(* CODESYS project simulacoes.project

Project tree, tasks and I/O mapping:
  Device : CODESYS Control Win V3, 3S - Smart Software Solutions GmbH, version 3.5.12.10
    application Application
      libraries: VisuDialogs, * (System); Util, * (System); Standard, * (System)
      task DefaultTask (cyclic, interval T#10ms, priority 16) calls PLC_PRG
      Data types/
      Global Variables/
        global variables ParafusosIOs
        global variables GVL
      POUs/
        program PLC_PRG [ST]
      Visualizations/
        visualisation tanque_DIG
        visualisation SILO
        visualisation semaforo
        visualisation garagem
        visualisation tanque_ANALOG
      trace Sampling_Trace (task ): 
      PROGRAMAS/
        garagem/
          program garagem_LD [LD]
          program garagem_ST [ST]
        tanqueD/
          program tanqueD_batelada [ST]
          program tanqueD_auto [ST]
          program tanqueD_main [ST]
          program tanqueD_manual [ST]
        silo/
          program silo_LD [LD]
          program silo_ST [ST]
        semaforo/
          program semaforo_LD [LD]
          program semaforo_ST [ST]
        tanqueA/
          program tanqueA_main [ST]
          function VOL_TO_LEVEL [ST]
          program tanqueA_process [ST]
          program tanqueA_manut [ST]
      SIMULADORES/
        program SIM_GARAGEM [LD]
        program SIM_SILO [LD]
        program SIMULADORES [ST]
        program SIM_TANQUE_DIG [LD]
        program SIM_TANQUE_ANALOG [LD]
      image pool ImagePool
      Symbols
  libraries: Standard, 3.5.12.0 (System); IecSfc, 3.4.2.0 (System); SysCallback23, 3.5.2.0 (System); VisuSymbols, 3.5.10.0 (System)
  GlobalImagePool
  text list GlobalTextList
  5ce3da45-db07-42e7-a21c-a00fff4ed8f6|semaforo\WALK2.bmp
*)

// Device/Application/Global Variables/ParafusosIOs
VAR_GLOBAL
// I/Os - SILO
	// Entradas digitais:
		xParBStartSilo	 :	BOOL;
		xParBStopSilo	 :	BOOL;
		xParChASilo		 :	BOOL;
		xParChBSilo		 :	BOOL;
		xParChCSilo		 :	BOOL;
		xParLevel				  :	BOOL;
		xParProx 				  :	BOOL;
	// Saídas digitais:
		xParRunSilo		 : BOOL;
		xParFillSilo	 : BOOL;
		xParFullSilo	 : BOOL;
		xParValve 		 : BOOL;
		xParMotor 		 : BOOL;

// I/Os - Semáforo
	// Entradas digitais:
		xParafBPedE 	 :	BOOL;
		xParafBPedD 	 :	BOOL;
	// Saídas digitais:
		xParafVermE 	 : BOOL;
		xParafVermD 	 : BOOL;
		xParafVerdE 	 : BOOL;
		xParafVerdD		 : BOOL;
		xParafAmarE 	 : BOOL;
		xParafAmarD 	 : BOOL;

// I/Os - Garagem
	// Entradas digitais:
		xParBOpen 		          :	BOOL;
		xParBClose 		 :	BOOL;
		xParBStopGar	 :	BOOL;
		xParLs1 		 		  :	BOOL;
		xParLs2 		  		  :	BOOL;
	// Saídas digitais:
		xParAjar		 : BOOL;
		xParOpen 		 : BOOL;
		xParShut 		 : BOOL;
		xParMotorUp 	 : BOOL;
		xParMotorDown	 : BOOL;

// I/Os - Tanque (Digital)
	// Entradas digitais:
		xParBStartTankD	 :	BOOL;
		xParBStopTankD	 :	BOOL;
		xParChATankD	 :	BOOL;
		xParChBTankD	 :	BOOL;
		xParChCTankD	 :	BOOL;
		xParFluxo1				  :	BOOL;
		xParFluxo2				  :	BOOL;
		xParFluxo3				  :	BOOL;
		xParTermostato			  :	BOOL;
		xParAltoD				  :	BOOL;
		xParBaixoD				  :	BOOL;
	// Saídas digitais:	
		xParBomba1D		 : BOOL;
		xParBomba2D		 : BOOL;
		xParBomba3D		 : BOOL;
		xParAquecD		 : BOOL;
		xParMistD		 : BOOL;
		xParRunTankD	 : BOOL;
		xParFullTankD	 : BOOL;
		xParIdleD		 : BOOL;

// I/Os - Tanque (Analógico)
	// Entradas digitais:
		xParBStartTankA	 :	BOOL;
		xParBStopTankA	 :	BOOL;
		xParChATankA	 :	BOOL;
		xParChBTankA	 :	BOOL;
		xParChCTankA	 :	BOOL;	
	// Entradas analógicas:
		iParSPB1				  :	INT;
		iParSPB2	 			  :	INT;
		iParSPTemp				  :	INT;
		iParUltras				  :	INT;
		iParTerm				  :	INT;
	// Saídas digitais:	
		xParBomba1A		 : BOOL;
		xParBomba2A		 : BOOL;
		xParBomba3A		 : BOOL;
		xParAquecA		 : BOOL;
		xParMistA		 : BOOL;
		xParRunTankA	 : BOOL;
		xParFullTankA	 : BOOL;
		xParIdleA		 : BOOL;
	// Saidas analógicas:	
		iParDisplayTemp    : INT;
		iParDisplayNivel   : INT;
END_VAR

// Device/Application/Global Variables/GVL
VAR_GLOBAL
	l1 : REAL := 2000.0;
	l2 : REAL := 5000.0;
	k : REAL := (10000.0/64.0); //Constante de conversão (litros/pulso)
	TankDMode : INT := 0;
	xEnableTankD : BOOL;
	LimTankD : REAL;
	xEnableTankA : BOOL;
	iTankAUnit : INT;
	TankAMode : INT := 0;
	rSupI1 : REAL;
	rSupI2 : REAL;
	rSupT : REAL;
	rTankALevel : REAL;
	rTankATemp : REAL;
	xTankARunning : BOOL;
	rTankASP1 : REAL;
	rTankASP2 : REAL;
	rTankASPTemp : REAL;
	allowStart : BOOL;
	LimTankA : REAL;
	blinkEnable : BOOL;
	blinkDuration : INT;
	tonoff : REAL;
	NULL : BOOL := FALSE;
	blinkTarget : POINTER TO BOOL := ADR(NULL);
	halfCicle : BOOL;
	heat : BOOL;
	LimTankAConv : REAL;
	capMax : REAL;
	defaultUnit : INT;
	rTankAVol : REAL;
	offset : REAL;
	batCont : INT := 0;
	prod : REAL := 0;
	processTarget : INT := 0;
	xEndLess : BOOL := TRUE;
	processID : INT;
	xstopAfterCurrent : BOOL;
	rTankDVol : REAL;
END_VAR

// Device/Application/POUs/PLC_PRG
PROGRAM PLC_PRG
VAR

END_VAR

SIMULADORES();
//garagem_LD();
garagem_ST();
//silo_LD();
silo_ST();
//semaforo_LD();
semaforo_ST();
tanqueD_main();
tanqueA_main();

END_PROGRAM

// Device/Application/SIMULADORES/SIMULADORES
PROGRAM SIMULADORES
VAR
END_VAR

SIM_GARAGEM();
SIM_SILO();
SIM_TANQUE_DIG();
SIM_TANQUE_ANALOG();

END_PROGRAM

// Device/Application/SIMULADORES/SIM_GARAGEM
PROGRAM SIM_GARAGEM
VAR
	portao		: 	RAMP_INT;
	porta		: 	INT;
	pin			: 	INT;
	T2g		: 	TON;
	T1g		: 	TON;
	fogo		: 	BOOL;
	fechado	: 	BOOL;
	aberto		: 	BOOL;
	Tfogo		: 	TON;
	fogosobe	: 	BOOL;
	fogodesce: 	BOOL;
	Pisca: BOOL;
	Pisca1: BLINK;
END_VAR
VAR // added by the converter: edge detectors and wires of the graphical bodies
    _w1 : USINT;
    _w2 : INT;
END_VAR

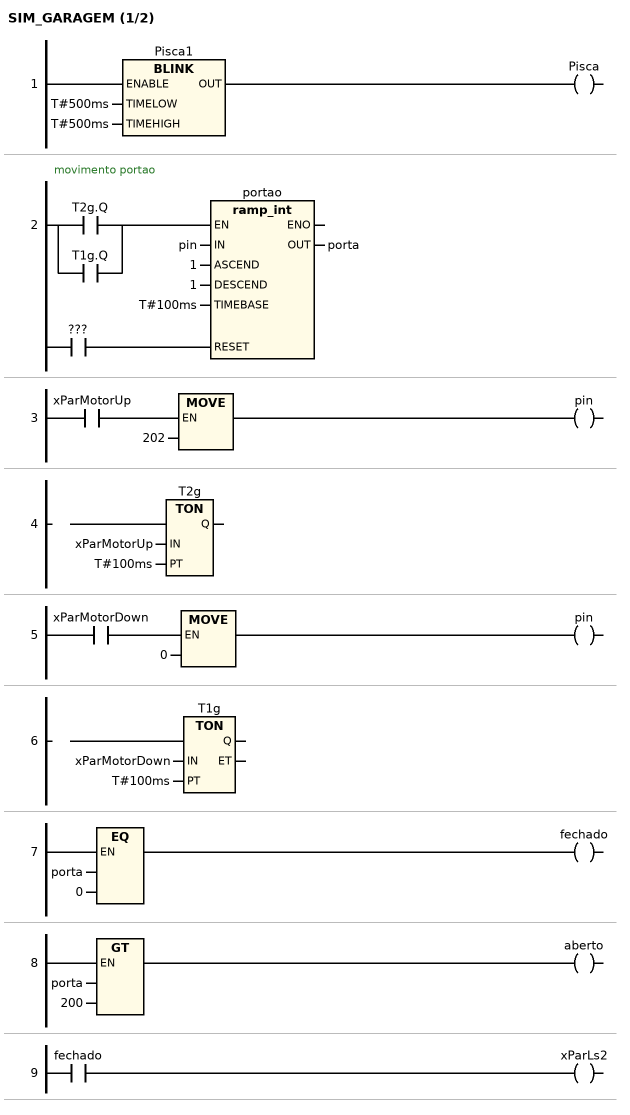
// NETWORK 1
Pisca1(ENABLE := TRUE, TIMELOW := T#500ms, TIMEHIGH := T#500ms); // BLINK
Pisca := Pisca1.OUT;

// NETWORK 2
// movimento portao
IF T2g.Q OR T1g.Q THEN
    portao(IN := pin, ASCEND := 1, DESCEND := 1, TIMEBASE := T#100ms, OUT => porta); // ramp_int
END_IF

// NETWORK 3
IF xParMotorUp THEN _w1 := 202; END_IF
pin := _w1;

// NETWORK 4
T2g(IN := xParMotorUp, PT := T#100ms); // TON

// NETWORK 5
IF xParMotorDown THEN _w2 := 0; END_IF
pin := _w2;

// NETWORK 6
T1g(IN := xParMotorDown, PT := T#100ms); // TON

// NETWORK 7
fechado := porta = 0;

// NETWORK 8
aberto := porta > 200;

// NETWORK 9
xParLs2 := fechado;

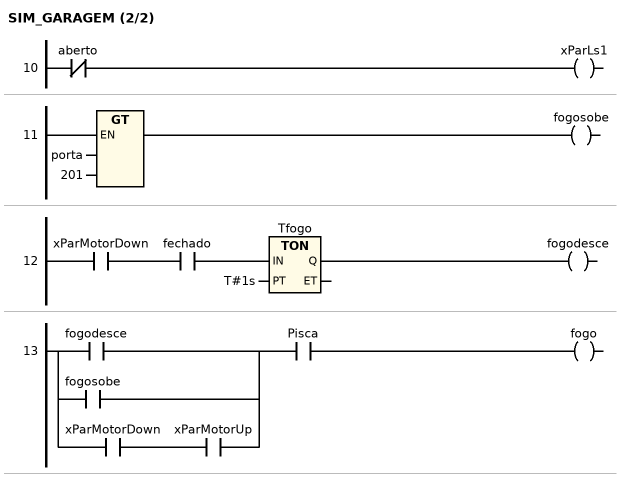
// NETWORK 10
xParLs1 := NOT aberto;

// NETWORK 11
fogosobe := porta > 201;

// NETWORK 12
Tfogo(IN := xParMotorDown AND fechado, PT := T#1s); // TON
fogodesce := Tfogo.Q;

// NETWORK 13
fogo := (fogodesce OR fogosobe OR xParMotorDown AND xParMotorUp) AND Pisca;

END_PROGRAM

// Device/Application/SIMULADORES/SIM_SILO
PROGRAM SIM_SILO
VAR
	aaux			: 	BOOL;
	Tcx				: 	TON;
	ccx				: 	CTU;
	resetesteira	: 	BOOL;
	caixa_mov1	: 	INT;
	caixa_mov		: 	INT;
	prox1			: 	BOOL;
	prox2			: 	BOOL;
	Tlevel			: 	TON;
	clevel			: 	CTU;
	level1			: 	INT;
	auxlevel		: 	BOOL;
	Talaga			: 	TON;
	calaga			: 	CTU;
	alaga			: 	INT;
	RESET		: 	BOOL;
	Pisca: BOOL;
	Pisca1: BLINK;
	CHEIA: BOOL;
END_VAR

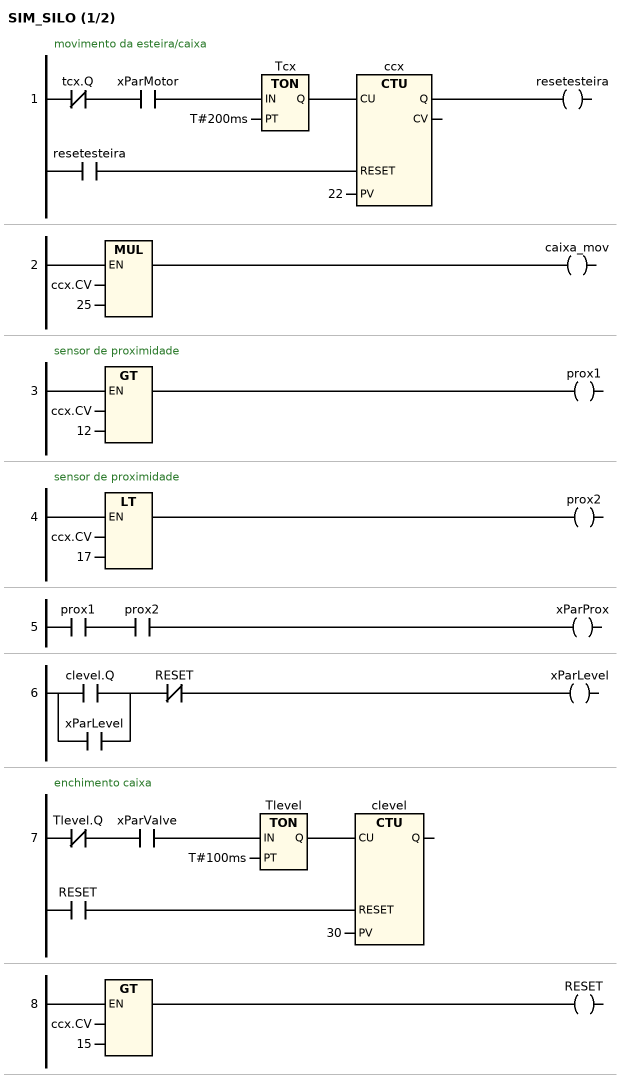
// NETWORK 1
// movimento da esteira/caixa
Tcx(IN := NOT tcx.Q AND xParMotor, PT := T#200ms); // TON
ccx(CU := Tcx.Q, RESET := resetesteira, PV := 22); // CTU
resetesteira := ccx.Q;

// NETWORK 2
caixa_mov := ccx.CV * 25;

// NETWORK 3
// sensor de proximidade
prox1 := ccx.CV > 12;

// NETWORK 4
// sensor de proximidade
prox2 := ccx.CV < 17;

// NETWORK 5
xParProx := prox1 AND prox2;

// NETWORK 6
xParLevel := (clevel.Q OR xParLevel) AND NOT RESET;

// NETWORK 7
// enchimento caixa
Tlevel(IN := NOT Tlevel.Q AND xParValve, PT := T#100ms); // TON
clevel(CU := Tlevel.Q, RESET := RESET, PV := 30); // CTU

// NETWORK 8
RESET := ccx.CV > 15;

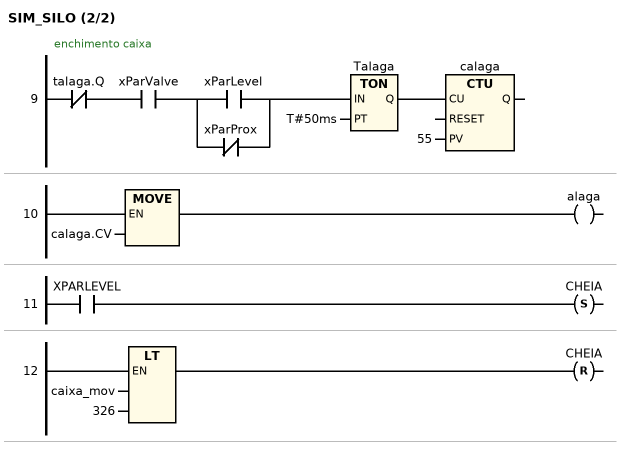
// NETWORK 9
// enchimento caixa
Talaga(IN := NOT talaga.Q AND xParValve AND (xParLevel OR NOT xParProx), PT := T#50ms); // TON
calaga(CU := Talaga.Q, PV := 55); // CTU

// NETWORK 10
alaga := calaga.CV;

// NETWORK 11
CHEIA S= XPARLEVEL;

// NETWORK 12
CHEIA R= caixa_mov < 326;

END_PROGRAM

// Device/Application/SIMULADORES/SIM_TANQUE_DIG
PROGRAM SIM_TANQUE_DIG
VAR
	CF1			: 	CTU;
	TF1			: 	TON;
	PB1			: 	BLINK;
	PF1			: 	BOOL :=0;
	TF2			: 	TON;
	CF2			: 	CTU;
	PB2			: 	BLINK;
	PF2			: 	BOOL :=0;
	TF3			: 	TON;
	CF3			: 	CTU;
	PB3			: 	BLINK;
	PF3			: 	BOOL :=0;
	NIVELAUX		: 	INT;
	PFOGO		: 	BLINK;
	PFIRE			: 	BOOL;
	PMIX			: 	BLINK;
	MIX1			: 	BOOL;
	tempadj		: 	INT;
	Tchama		: 	TON;
	chamaup		: 	BOOL;
	chamadown	: 	BOOL;
	chamafall		: 	F_TRIG;
	chamaload	: 	BOOL;
	Cchama		: 	CTUD;
	NIVELAUX2	: 	BOOL;
	bombafogo	: 	BOOL;
	TRANSB		: 	TON;
	CTRANSB		: 	CTU;
	NIVELAUX3	: 	BOOL;
	nivelCM: INT;
	Tfogo2: TON;
	Pisca: BOOL;
	Pisca1: BLINK;
	PBfogo: BLINK;
	TON_0: TOF;
END_VAR
VAR // added by the converter: edge detectors and wires of the graphical bodies
    _w1 : INT;
END_VAR

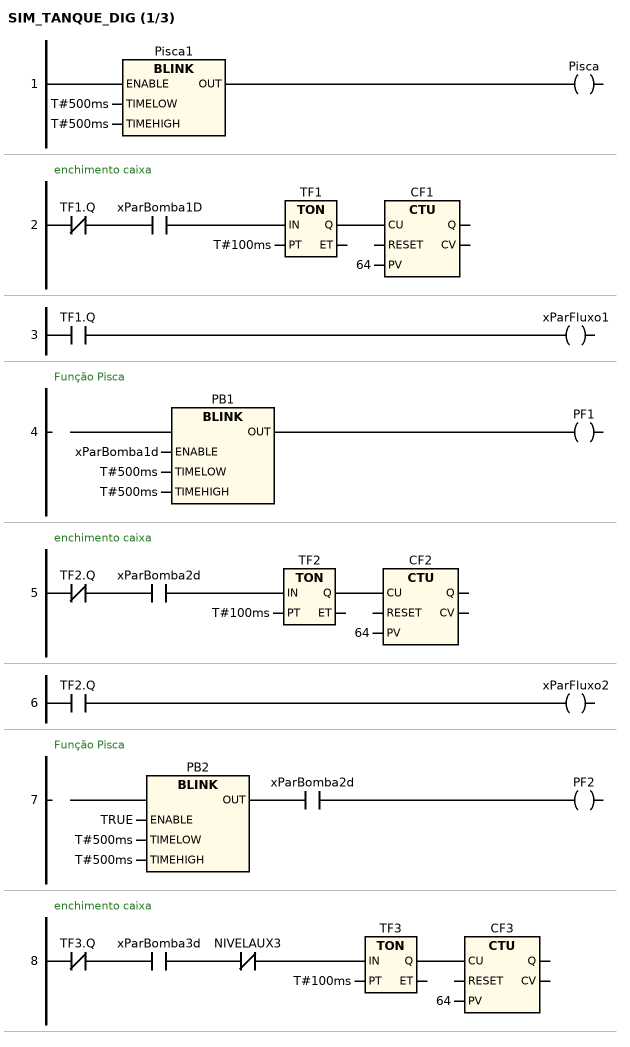
// NETWORK 1
Pisca1(ENABLE := TRUE, TIMELOW := T#500ms, TIMEHIGH := T#500ms); // BLINK
Pisca := Pisca1.OUT;

// NETWORK 2
// enchimento caixa
TF1(IN := NOT TF1.Q AND xParBomba1D, PT := T#100ms); // TON
CF1(CU := TF1.Q, PV := 64); // CTU

// NETWORK 3
xParFluxo1 := TF1.Q;

// NETWORK 4
// Função Pisca
PB1(ENABLE := xParBomba1d, TIMELOW := T#500ms, TIMEHIGH := T#500ms); // BLINK
PF1 := PB1.OUT;

// NETWORK 5
// enchimento caixa
TF2(IN := NOT TF2.Q AND xParBomba2d, PT := T#100ms); // TON
CF2(CU := TF2.Q, PV := 64); // CTU

// NETWORK 6
xParFluxo2 := TF2.Q;

// NETWORK 7
// Função Pisca
PB2(ENABLE := TRUE, TIMELOW := T#500ms, TIMEHIGH := T#500ms); // BLINK
PF2 := PB2.OUT AND xParBomba2d;

// NETWORK 8
// enchimento caixa
TF3(IN := NOT TF3.Q AND xParBomba3d AND NOT NIVELAUX3, PT := T#100ms); // TON
CF3(CU := TF3.Q, PV := 64); // CTU

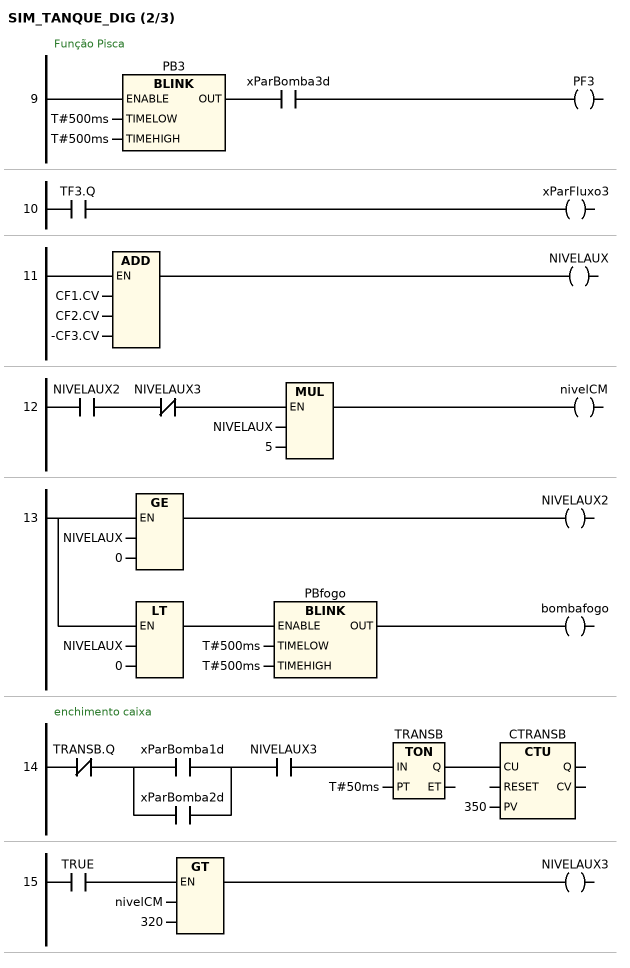
// NETWORK 9
// Função Pisca
PB3(ENABLE := TRUE, TIMELOW := T#500ms, TIMEHIGH := T#500ms); // BLINK
PF3 := PB3.OUT AND xParBomba3d;

// NETWORK 10
xParFluxo3 := TF3.Q;

// NETWORK 11
NIVELAUX := CF1.CV + CF2.CV + (-CF3.CV);

// NETWORK 12
IF NIVELAUX2 AND NOT NIVELAUX3 THEN _w1 := NIVELAUX * 5; END_IF
nivelCM := _w1;

// NETWORK 13
NIVELAUX2 := NIVELAUX >= 0;
PBfogo(ENABLE := NIVELAUX < 0, TIMELOW := T#500ms, TIMEHIGH := T#500ms); // BLINK
bombafogo := PBfogo.OUT;

// NETWORK 14
// enchimento caixa
TRANSB(IN := NOT TRANSB.Q AND (xParBomba1d OR xParBomba2d) AND NIVELAUX3, PT := T#50ms); // TON
CTRANSB(CU := TRANSB.Q, PV := 350); // CTU

// NETWORK 15
NIVELAUX3 := nivelCM > 320;

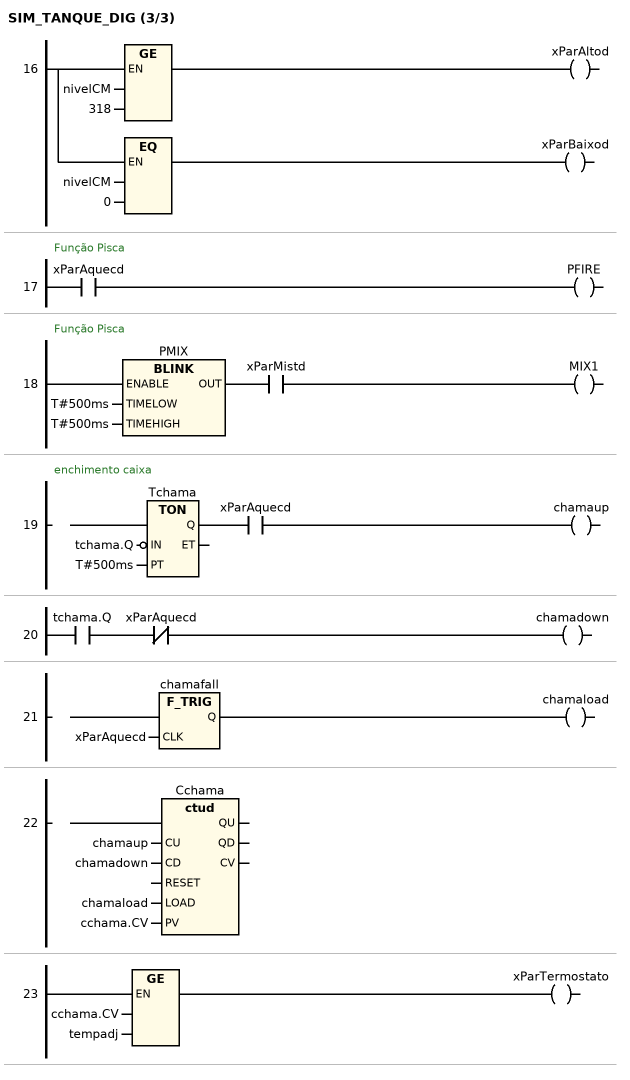
// NETWORK 16
xParAltod := nivelCM >= 318;
xParBaixod := nivelCM = 0;

// NETWORK 17
// Função Pisca
PFIRE := xParAquecd;

// NETWORK 18
// Função Pisca
PMIX(ENABLE := TRUE, TIMELOW := T#500ms, TIMEHIGH := T#500ms); // BLINK
MIX1 := PMIX.OUT AND xParMistd;

// NETWORK 19
// enchimento caixa
Tchama(IN := NOT tchama.Q, PT := T#500ms); // TON
chamaup := Tchama.Q AND xParAquecd;

// NETWORK 20
chamadown := tchama.Q AND NOT xParAquecd;

// NETWORK 21
chamafall(CLK := xParAquecd); // F_TRIG
chamaload := chamafall.Q;

// NETWORK 22
Cchama(CU := chamaup, CD := chamadown, LOAD := chamaload, PV := cchama.CV); // ctud

// NETWORK 23
xParTermostato := cchama.CV >= tempadj;

END_PROGRAM

// Device/Application/SIMULADORES/SIM_TANQUE_ANALOG
PROGRAM SIM_TANQUE_ANALOG
VAR
	CF1			: 	CTU;
	TF1			: 	TON;
	PB1			: 	BLINK;
	PF1			: 	BOOL :=0;
	TF2			: 	TON;
	CF2			: 	CTU;
	PB2			: 	BLINK;
	PF2			: 	BOOL :=0;
	TF3			: 	TON;
	CF3			: 	CTU;
	PB3			: 	BLINK;
	PF3			: 	BOOL :=0;
	NIVELAUX		: 	INT;
	PFOGO		: 	BLINK;
	PFIRE			: 	BOOL;
	PMIX			: 	BLINK;
	MIX1			: 	BOOL;
	tempadj		: 	INT;
	Tchama		: 	TON;
	chamaup		: 	BOOL;
	chamadown	: 	BOOL;
	chamafall		: 	F_TRIG;
	chamaload	: 	BOOL;
	Cchama		: 	CTUD;
	NIVELAUX2	: 	BOOL;
	bombafogo	: 	BOOL;
	TRANSB		: 	TON;
	CTRANSB		: 	CTU;
	NIVELAUX3	: 	BOOL;
	nivelCM: INT;
	Tfogo2: TON;
	Pisca: BOOL;
	Pisca1: BLINK;
	PBfogo: BLINK;
	TON_0: TOF;
	TEMP_SCALE: LIN_TRAFO;
	TEMPAUX: REAL;
	NIVEL_SCALE: LIN_TRAFO;
	NIVEL_INT: REAL;
	RAMPANIVEL: ramp_int;
	PIN : INT;
	TON_1: TON;
	spbomba1: LIN_TRAFO;
	setbomba1 : INT;
	setbomba2 : INT;
	settemp : INT;
	spbomba2: LIN_TRAFO;
	spointtemp: LIN_TRAFO;
END_VAR
VAR // added by the converter: edge detectors and wires of the graphical bodies
    _w1, _w2 : INT;
END_VAR

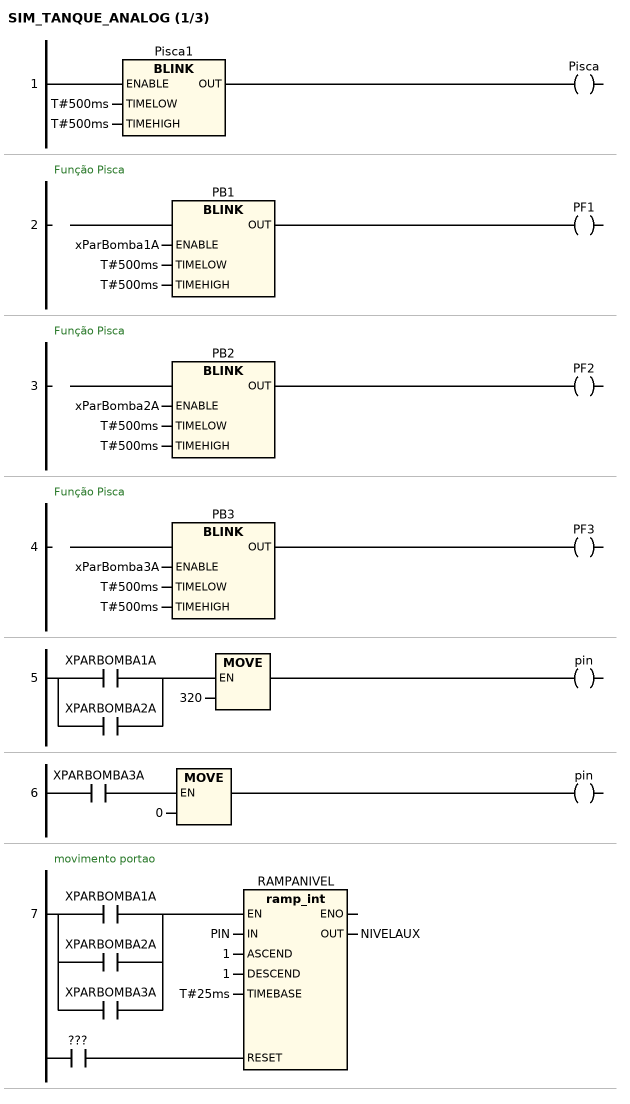
// NETWORK 1
Pisca1(ENABLE := TRUE, TIMELOW := T#500ms, TIMEHIGH := T#500ms); // BLINK
Pisca := Pisca1.OUT;

// NETWORK 2
// Função Pisca
PB1(ENABLE := xParBomba1A, TIMELOW := T#500ms, TIMEHIGH := T#500ms); // BLINK
PF1 := PB1.OUT;

// NETWORK 3
// Função Pisca
PB2(ENABLE := xParBomba2A, TIMELOW := T#500ms, TIMEHIGH := T#500ms); // BLINK
PF2 := PB2.OUT;

// NETWORK 4
// Função Pisca
PB3(ENABLE := xParBomba3A, TIMELOW := T#500ms, TIMEHIGH := T#500ms); // BLINK
PF3 := PB3.OUT;

// NETWORK 5
IF XPARBOMBA1A OR XPARBOMBA2A THEN _w1 := 320; END_IF
pin := _w1;

// NETWORK 6
IF XPARBOMBA3A THEN _w2 := 0; END_IF
pin := _w2;

// NETWORK 7
// movimento portao
IF XPARBOMBA1A OR XPARBOMBA2A OR XPARBOMBA3A THEN
    RAMPANIVEL(IN := PIN, ASCEND := 1, DESCEND := 1, TIMEBASE := T#25ms, OUT => NIVELAUX); // ramp_int
END_IF

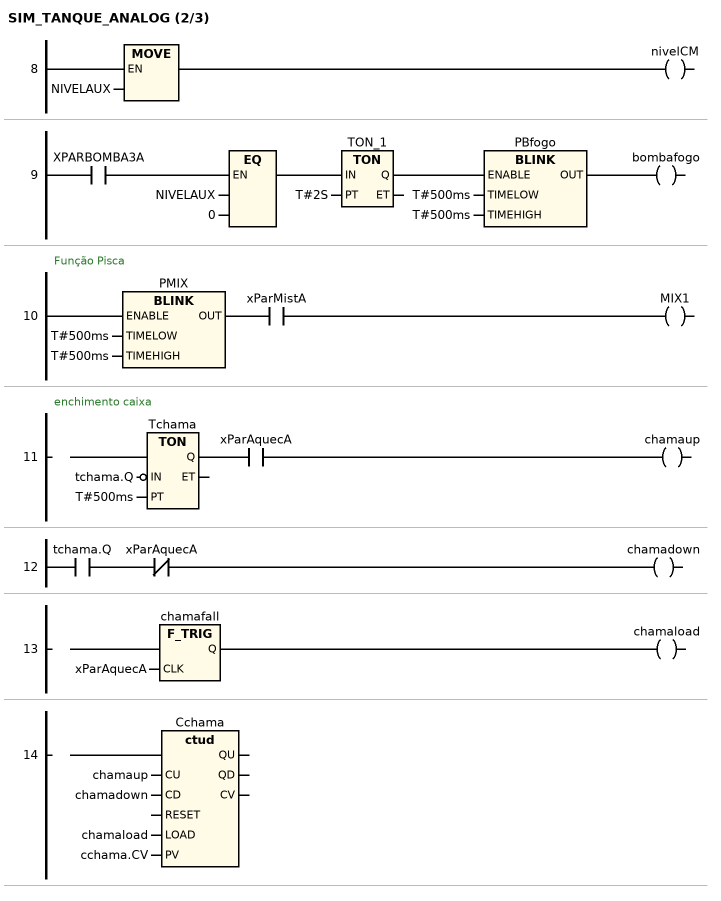
// NETWORK 8
nivelCM := NIVELAUX;

// NETWORK 9
TON_1(IN := XPARBOMBA3A AND NIVELAUX = 0, PT := T#2S); // TON
PBfogo(ENABLE := TON_1.Q, TIMELOW := T#500ms, TIMEHIGH := T#500ms); // BLINK
bombafogo := PBfogo.OUT;

// NETWORK 10
// Função Pisca
PMIX(ENABLE := TRUE, TIMELOW := T#500ms, TIMEHIGH := T#500ms); // BLINK
MIX1 := PMIX.OUT AND xParMistA;

// NETWORK 11
// enchimento caixa
Tchama(IN := NOT tchama.Q, PT := T#500ms); // TON
chamaup := Tchama.Q AND xParAquecA;

// NETWORK 12
chamadown := tchama.Q AND NOT xParAquecA;

// NETWORK 13
chamafall(CLK := xParAquecA); // F_TRIG
chamaload := chamafall.Q;

// NETWORK 14
Cchama(CU := chamaup, CD := chamadown, LOAD := chamaload, PV := cchama.CV); // ctud

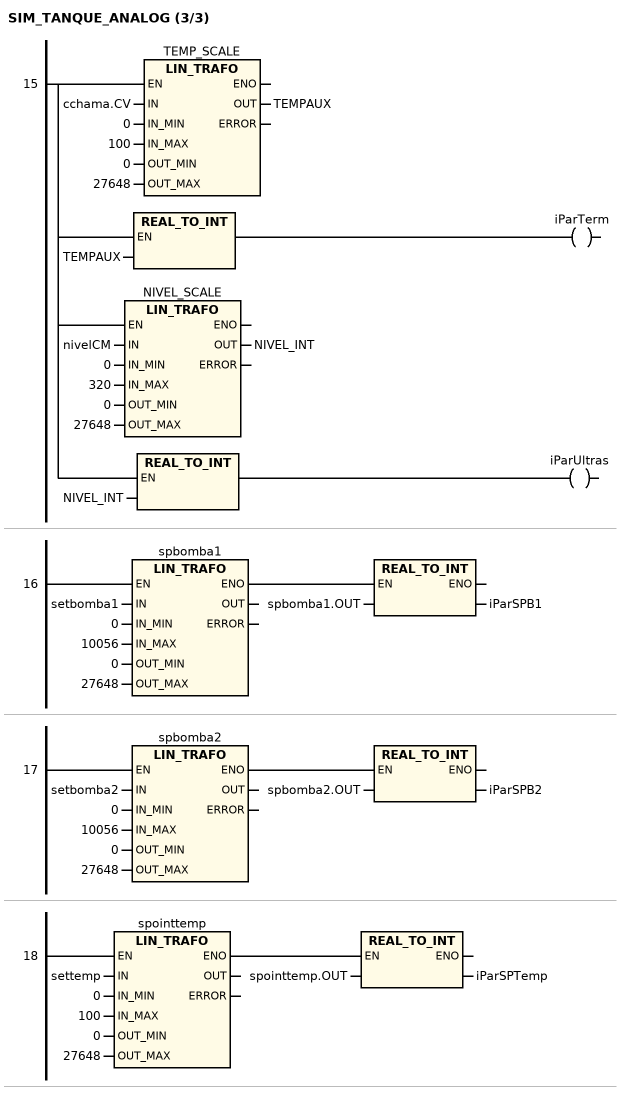
// NETWORK 15
TEMP_SCALE(IN := cchama.CV, IN_MIN := 0, IN_MAX := 100, OUT_MIN := 0, OUT_MAX := 27648, OUT => TEMPAUX); // LIN_TRAFO
iParTerm := REAL_TO_INT(TEMPAUX);
NIVEL_SCALE(IN := nivelCM, IN_MIN := 0, IN_MAX := 320, OUT_MIN := 0, OUT_MAX := 27648, OUT => NIVEL_INT); // LIN_TRAFO
iParUltras := REAL_TO_INT(NIVEL_INT);

// NETWORK 16
spbomba1(IN := setbomba1, IN_MIN := 0, IN_MAX := 10056, OUT_MIN := 0, OUT_MAX := 27648); // LIN_TRAFO
iParSPB1 := REAL_TO_INT(spbomba1.OUT);

// NETWORK 17
spbomba2(IN := setbomba2, IN_MIN := 0, IN_MAX := 10056, OUT_MIN := 0, OUT_MAX := 27648); // LIN_TRAFO
iParSPB2 := REAL_TO_INT(spbomba2.OUT);

// NETWORK 18
spointtemp(IN := settemp, IN_MIN := 0, IN_MAX := 100, OUT_MIN := 0, OUT_MAX := 27648); // LIN_TRAFO
iParSPTemp := REAL_TO_INT(spointtemp.OUT);

END_PROGRAM

// Device/Application/PROGRAMAS/garagem/garagem_LD
PROGRAM garagem_LD
VAR
END_VAR
VAR // added by the converter: edge detectors and wires of the graphical bodies
    _w1, _w2, _w3 : BOOL;
END_VAR

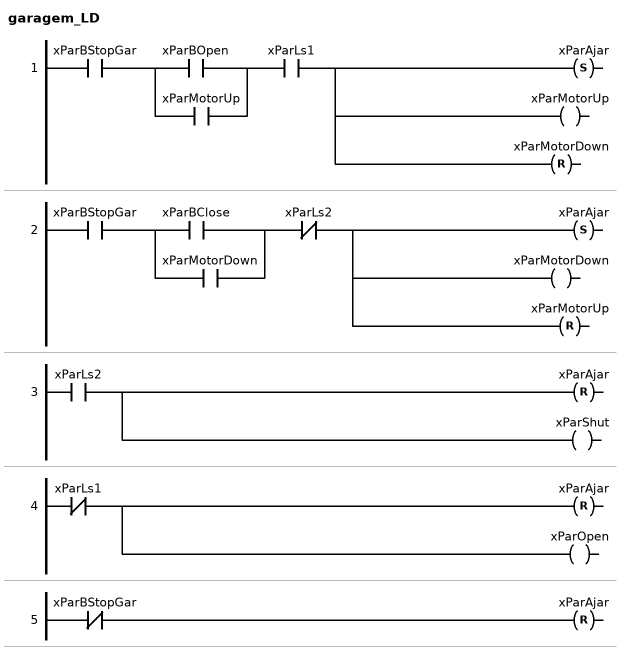
// NETWORK 1
_w1 := xParBStopGar AND (xParBOpen OR xParMotorUp) AND xParLs1;
xParAjar S= _w1;
xParMotorUp := _w1;
xParMotorDown R= _w1;

// NETWORK 2
_w2 := xParBStopGar AND (xParBClose OR xParMotorDown) AND NOT xParLs2;
xParAjar S= _w2;
xParMotorDown := _w2;
xParMotorUp R= _w2;

// NETWORK 3
xParAjar R= xParLs2;
xParShut := xParLs2;

// NETWORK 4
_w3 := NOT xParLs1;
xParAjar R= _w3;
xParOpen := _w3;

// NETWORK 5
xParAjar R= NOT xParBStopGar;

END_PROGRAM

// Device/Application/PROGRAMAS/garagem/garagem_ST
PROGRAM garagem_ST
VAR
END_VAR

//Condição de stop:
IF NOT xParBStopGar THEN
	xParMotorUp := FALSE;
	xParMotorDown := FALSE;
END_IF

//Acionamento dos motores pelas botoeiras:
IF xParBOpen THEN
	xParMotorUp := TRUE;
	xParMotorDown := FALSE;
END_IF
IF xParBClose THEN
	xParMotorUp := FALSE;
	xParMotorDown := TRUE;
END_IF

//Desligamento aotumático pelos fim-de-curso:
IF NOT xParLs1 THEN
	xParMotorUp := FALSE;
END_IF
IF xParLs2 THEN
	xParMotorDown := FALSE;
END_IF

//Lâmpadas:
xParAjar := xParMotorUp OR xParMotorDown;
xParOpen := NOT xParLs1;
xParShut := xParLs2;

END_PROGRAM

// Device/Application/PROGRAMAS/silo/silo_LD
PROGRAM silo_LD
VAR
	running: BOOL;
	fill: BOOL;
	full: BOOL;
END_VAR
VAR // added by the converter: edge detectors and wires of the graphical bodies
    _w1, _w2, _w3, _w4 : BOOL;
END_VAR

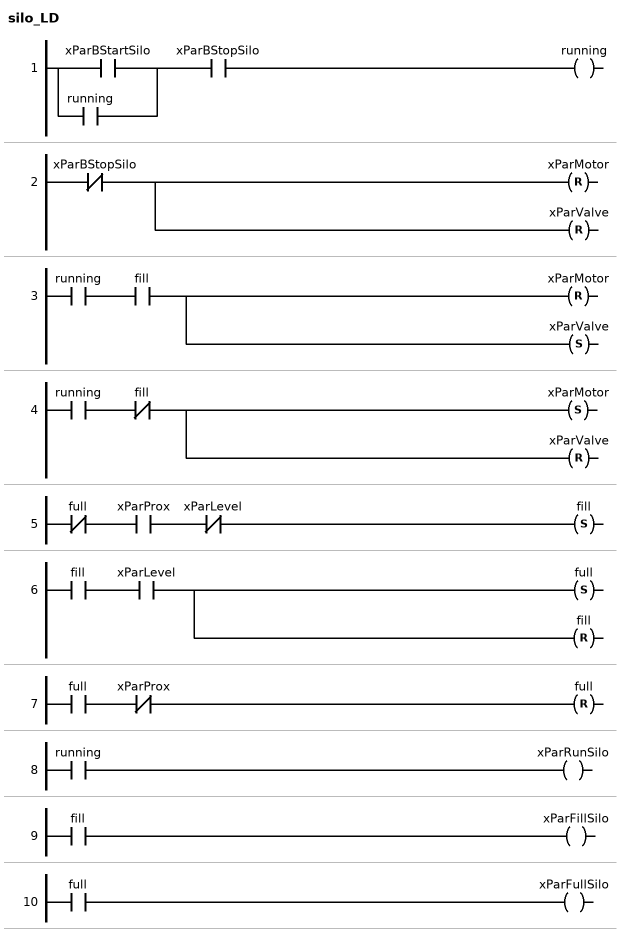
// NETWORK 1
running := (xParBStartSilo OR running) AND xParBStopSilo;

// NETWORK 2
_w1 := NOT xParBStopSilo;
xParMotor R= _w1;
xParValve R= _w1;

// NETWORK 3
_w2 := running AND fill;
xParMotor R= _w2;
xParValve S= _w2;

// NETWORK 4
_w3 := running AND NOT fill;
xParMotor S= _w3;
xParValve R= _w3;

// NETWORK 5
fill S= NOT full AND xParProx AND NOT xParLevel;

// NETWORK 6
_w4 := fill AND xParLevel;
full S= _w4;
fill R= _w4;

// NETWORK 7
full R= full AND NOT xParProx;

// NETWORK 8
xParRunSilo := running;

// NETWORK 9
xParFillSilo := fill;

// NETWORK 10
xParFullSilo := full;

END_PROGRAM

// Device/Application/PROGRAMAS/silo/silo_ST
PROGRAM silo_ST
VAR
	estado : INT := 0;
	run : BOOL := FALSE;
END_VAR

IF run THEN
	//Definição dos estados:
	IF estado = 1 THEN
		xParValve := FALSE;
		xParMotor := TRUE;
		xParRunSilo := TRUE;
		xParFillSilo := FALSE;
		xParFullSilo := FALSE;
		//Condição de mudança de estado:
		IF xParProx THEN
			estado := 2;
		END_IF
	END_IF
	IF estado = 2 THEN
		xParValve := TRUE;
		xParMotor := FALSE;
		xParRunSilo := TRUE;
		xParFillSilo := TRUE;
		xParFullSilo := FALSE;
		//Condição de mudança de estado:
		IF xParLevel THEN
			estado := 3;
		END_IF
	END_IF
	IF estado = 3 THEN
		xParValve := FALSE;
		xParMotor := TRUE;
		xParRunSilo := TRUE;
		xParFillSilo := FALSE;
		xParFullSilo := TRUE;
		//Condição de reinício do ciclo:
		IF NOT xParProx THEN
			estado := 1;
		END_IF
	END_IF
END_IF


//Condições para início do ciclo:
IF xParBStartSilo THEN
	run := TRUE;
	IF NOT INT_TO_BOOL(estado) THEN
		estado := 1;
	END_IF
END_IF

//Condição de STOP:
IF NOT xParBStopSilo THEN
	run := FALSE;
	xParValve := FALSE;
		xParMotor := FALSE;
		xParRunSilo := FALSE;
		xParFillSilo := FALSE;
		xParFullSilo := FALSE;
END_IF

END_PROGRAM

// Device/Application/PROGRAMAS/semaforo/semaforo_LD
PROGRAM semaforo_LD
VAR
	VdD: TON;
	AmD: TON;
	VdE: TON;
	AmE: TON;
	reset: BOOL;
END_VAR

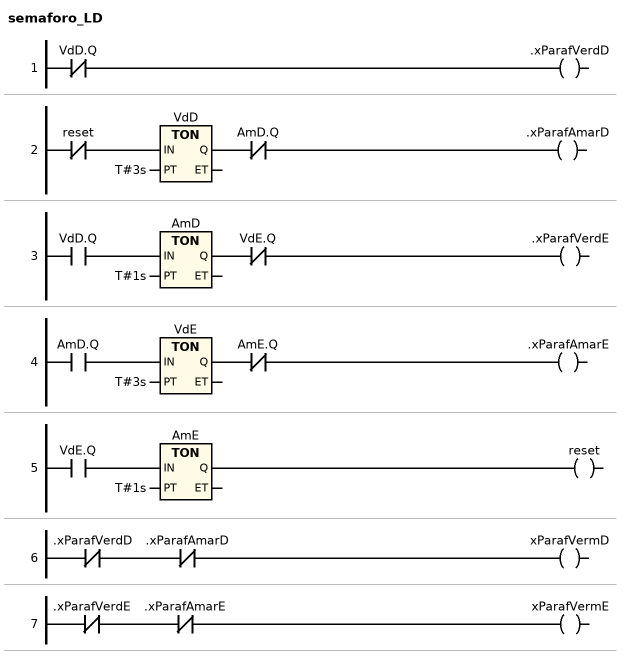
// NETWORK 1
.xParafVerdD := NOT VdD.Q;

// NETWORK 2
VdD(IN := NOT reset, PT := T#3s); // TON
.xParafAmarD := VdD.Q AND NOT AmD.Q;

// NETWORK 3
AmD(IN := VdD.Q, PT := T#1s); // TON
.xParafVerdE := AmD.Q AND NOT VdE.Q;

// NETWORK 4
VdE(IN := AmD.Q, PT := T#3s); // TON
.xParafAmarE := VdE.Q AND NOT AmE.Q;

// NETWORK 5
AmE(IN := VdE.Q, PT := T#1s); // TON
reset := AmE.Q;

// NETWORK 6
xParafVermD := NOT .xParafVerdD AND NOT .xParafAmarD;

// NETWORK 7
xParafVermE := NOT .xParafVerdE AND NOT .xParafAmarE;

END_PROGRAM

// Device/Application/PROGRAMAS/semaforo/semaforo_ST
PROGRAM semaforo_ST
VAR
	TIMER : TON;
	enable : BOOL := TRUE;
	sec: REAL;
END_VAR

//Lógica de contagem incremental temporizada resetável:
IF TIMER.Q THEN
	enable := FALSE;
END_IF
TIMER(IN := enable, PT := T#12S);
IF NOT enable THEN
	enable := TRUE;
END_IF

//Variável auxiliar para facilitar a conversão e comparação:
sec := TIME_TO_REAL(TIMER.ET);

//Lógica semáforo esquerda:
IF sec < 7E3 THEN
	xParafAmarE := FALSE;
	xParafVermE := TRUE;
END_IF
IF (sec > 7E3) AND (sec < 10E3) THEN
	xParafVermE := FALSE;
	xParafVerdE := TRUE;	
END_IF
IF sec > 10E3 THEN
	xParafVerdE := FALSE;
	xParafAmarE := TRUE;
END_IF

//Lógica semáforo direita:
IF (sec < 1E3) OR (sec > 6E3) THEN
	xParafAmarD := FALSE;
	xParafVermD := TRUE;
END_IF
IF (sec > 1E3) AND (sec < 4E3) THEN
	xParafVermD := FALSE;
	xParafVerdD := TRUE;	
END_IF
IF (sec > 4E3) AND (sec < 6E3) THEN
	xParafVerdD := FALSE;
	xParafAmarD := TRUE;
END_IF

END_PROGRAM

// Device/Application/PROGRAMAS/tanqueD/tanqueD_main
PROGRAM tanqueD_main
VAR
END_VAR

//Verifica prioridade do transitório:
IF NOT xEnableTankD THEN
	IF xParChATankD THEN
		//Modo automático:
		TankDMode := 1;
	ELSE
		IF xParChBTankD THEN
			//Batelada:
			TankDMode := 2;
		ELSE
			IF xParChCTankD THEN
				//Manual:
				TankDMode := 3;
			ELSE
				TankDMode := 0;
			END_IF
		END_IF
	END_IF	
END_IF

CASE TankDMode OF
	1:	tanqueD_auto();
	2:	tanqueD_batelada();
	3:	tanqueD_manual();
END_CASE

//Limite para o segundo ingrediente:
LimTankD := 10000-l1;

END_PROGRAM

// Device/Application/PROGRAMAS/tanqueD/tanqueD_auto
PROGRAM tanqueD_auto
VAR
	mctr : TOF;
	pulses1 : CTU;
	pulses2 : CTU;
	pulses3 : CTU;
	resetp1 : BOOL;
	resetp2 : BOOL;
	resetp3 : BOOL;
	running : BOOL;
	mix : BOOL;
	state : INT;
END_VAR

//Declaração do timer de desligamento da mistura:
mctr(IN:=mix, PT:=T#5S);

//Declaração os contadores de fluxo:
pulses1(CU:=xParFluxo1, RESET:=resetp1, PV:=REAL_TO_WORD(l1/k));
pulses2(CU:=xParFluxo2, RESET:=resetp2, PV:=REAL_TO_WORD(l2/k));
pulses3(CU:=xParFluxo3, RESET:=resetp3, PV:=REAL_TO_WORD((l1+l2)/k));

//Condição de início do ciclo:
IF xParBStartTankD THEN
	running := TRUE;
	IF state=0 THEN
		state := 1;
	END_IF
END_IF

//Escolha de estado:
IF running THEN
	CASE state OF
		//Adiciona os ingredientes:	
		1:	IF pulses1.Q AND pulses2.Q THEN
				resetp1 := TRUE;
				resetp2 := TRUE;
				state := 2;
			ELSE
				rTankDVol := ((pulses1.CV + pulses2.CV)*k);
				resetp1 := FALSE;
				resetp2 := FALSE;
			END_IF	
			IF pulses1.Q THEN
				xParBomba1D := FALSE;
			ELSE
				xParBomba1D := TRUE;
			END_IF
			IF pulses2.Q THEN
				xParBomba2D := FALSE;
			ELSE
				xParBomba2D := TRUE;
			END_IF
		//Aquece e mistura:
		2:	xParAquecD := TRUE;
			mix := TRUE;
			IF xParTermostato THEN
				xParAquecD := FALSE;
				mix := FALSE;
				state := 3;
			END_IF
			xParMistD := mctr.Q;
		//Aguarda mistura:
		3:	xParMistD := mctr.Q;
			IF NOT mctr.Q THEN
				state := 4;
			END_IF
		//Esvazia o tanque:
		4: IF pulses3.Q THEN
				xParBomba3D := FALSE;
				resetp3 := TRUE;
				state := 1;
			ELSE
				rTankDVol := (l1+l2-(pulses3.CV*k));
				xParBomba3D := TRUE;
				resetp3:= FALSE;
			END_IF
	END_CASE
	
	//Indicações:
	xParRunTankD := running;
	IF state=2 OR state=3 THEN
		xParFullTankD := TRUE;
	ELSE
		xParFullTankD := FALSE;
	END_IF
	IF state=2 THEN
		xParIdleD := TRUE;
	ELSE
		xParIdleD := FALSE;
	END_IF
END_IF

//Condição de parada do oiclo:
IF NOT xParBStopTankD THEN
	running := FALSE;
	xParBomba1D := FALSE;
	xParBomba2D := FALSE;
	xParBomba3D := FALSE;
	xParAquecD := FALSE;
	xParMistD := FALSE;
	xParRunTankD := FALSE;
	xParFullTankD := FALSE;
	xParIdleD := FALSE;
END_IF

END_PROGRAM

// Device/Application/PROGRAMAS/tanqueD/tanqueD_batelada
PROGRAM tanqueD_batelada
VAR
	mctr : TOF;
	pulses1 : CTU;
	pulses2 : CTU;
	pulses3 : CTU;
	resetp1 : BOOL;
	resetp2 : BOOL;
	resetp3 : BOOL;
	running : BOOL;
	mix : BOOL;
	state : INT;
END_VAR

//Declaração do timer de desligamento da mistura:
mctr(IN:=mix, PT:=T#5S);

//Declaração os contadores de fluxo:
pulses1(CU:=xParFluxo1, RESET:=resetp1, PV:=REAL_TO_WORD(l1/k));
pulses2(CU:=xParFluxo2, RESET:=resetp2, PV:=REAL_TO_WORD(l2/k));
pulses3(CU:=xParFluxo3, RESET:=resetp3, PV:=REAL_TO_WORD((l1+l2)/k));

//Condição de início do ciclo:
IF xParBStartTankD THEN
	running := TRUE;
	IF state=0 THEN
		state := 1;
	END_IF
END_IF

//Condição de parada do oiclo:
IF NOT xParBStopTankD THEN
	running := FALSE;
END_IF

//Escolha de estado:
IF running THEN
	CASE state OF
		//Adiciona os ingredientes:	
		1:	IF pulses1.Q AND pulses2.Q THEN
				resetp1 := TRUE;
				resetp2 := TRUE;
				state := 2;
			ELSE
				rTankDVol := ((pulses1.CV + pulses2.CV)*k);
				resetp1 := FALSE;
				resetp2 := FALSE;
			END_IF	
			IF pulses1.Q THEN
				xParBomba1D := FALSE;
			ELSE
				xParBomba1D := TRUE;
			END_IF
			IF pulses2.Q THEN
				xParBomba2D := FALSE;
			ELSE
				xParBomba2D := TRUE;
			END_IF
		//Aquece e mistura:
		2:	xParAquecD := TRUE;
			mix := TRUE;
			IF xParTermostato THEN
				xParAquecD := FALSE;
				mix := FALSE;
				state := 3;
			END_IF
			xParMistD := mctr.Q;
		//Aguarda mistura:
		3:	xParMistD := mctr.Q;
			IF NOT mctr.Q THEN
				state := 4;
			END_IF
		//Esvazia o tanque:
		4: IF pulses3.Q THEN
				xParBomba3D := FALSE;
				resetp3 := TRUE;
				running:= FALSE;
				state := 0;
				rTankDVol := 0;
			ELSE
				rTankDVol := (l1+l2-(pulses3.CV*k));
				xParBomba3D := TRUE;
				resetp3:= FALSE;
			END_IF
	END_CASE
	
	//Indicações:
	xParRunTankD := running;
	IF state=2 OR state=3 THEN
		xParFullTankD := TRUE;
	ELSE
		xParFullTankD := FALSE;
	END_IF
	IF state=2 THEN
		xParIdleD := TRUE;
	ELSE
		xParIdleD := FALSE;
	END_IF
END_IF

//Desligando saídas na parada::
IF NOT running THEN
	xParBomba1D := FALSE;
	xParBomba2D := FALSE;
	xParBomba3D := FALSE;
	xParAquecD := FALSE;
	xParMistD := FALSE;
	xParRunTankD := FALSE;
	xParFullTankD := FALSE;
	xParIdleD := FALSE;
END_IF

END_PROGRAM

// Device/Application/PROGRAMAS/tanqueD/tanqueD_manual
PROGRAM tanqueD_manual
VAR
	mctr : TOF;
	pulses1 : CTU;
	pulses2 : CTU;
	pulses3 : CTU;
	resetp1 : BOOL;
	resetp2 : BOOL;
	resetp3 : BOOL;
	running : BOOL;
	mix : BOOL;
	state : INT;
	k : REAL := (10000.0/64.0); //Constante de conversão (litros/pulso)
END_VAR

//Declaração do timer de desligamento da mistura:
mctr(IN:=mix, PT:=T#5S);

//Declaração os contadores de fluxo:
pulses1(CU:=xParFluxo1, RESET:=resetp1, PV:=REAL_TO_WORD(l1/k));
pulses2(CU:=xParFluxo2, RESET:=resetp2, PV:=REAL_TO_WORD(l2/k));
pulses3(CU:=xParFluxo3, RESET:=resetp3, PV:=REAL_TO_WORD((l1+l2)/k));

//Condição de início do ciclo:
IF xParBStartTankD THEN
	running := TRUE;
	IF state=0 THEN
		state := 1;
	END_IF
END_IF

//Escolha de estado:
IF running THEN
	CASE state OF
		//Adiciona os ingredientes:	
		1:	IF pulses1.Q AND pulses2.Q THEN
				resetp1 := TRUE;
				resetp2 := TRUE;
				state := 2;
			ELSE
				resetp1 := FALSE;
				resetp2 := FALSE;
			END_IF	
			IF pulses1.Q THEN
				xParBomba1D := FALSE;
			ELSE
				xParBomba1D := TRUE;
			END_IF
			IF pulses2.Q THEN
				xParBomba2D := FALSE;
			ELSE
				xParBomba2D := TRUE;
			END_IF
		//Aquece e mistura:
		2:	xParAquecD := TRUE;
			mix := TRUE;
			IF xParTermostato THEN
				xParAquecD := FALSE;
				mix := FALSE;
				state := 3;
			END_IF
			xParMistD := mctr.Q;
		//Aguarda mistura:
		3:	xParMistD := mctr.Q;
			IF NOT mctr.Q THEN
				state := 4;
			END_IF
		//Esvazia o tanque:
		4: IF pulses3.Q THEN
				xParBomba3D := FALSE;
				resetp3 := TRUE;
				state := 1;
			ELSE
				xParBomba3D := TRUE;
				resetp3:= FALSE;
			END_IF
	END_CASE
	
	//Indicações:
	xParRunTankD := running;
	IF state=2 OR state=3 THEN
		xParFullTankD := TRUE;
	ELSE
		xParFullTankD := FALSE;
	END_IF
	IF state=2 THEN
		xParIdleD := TRUE;
	ELSE
		xParIdleD := FALSE;
	END_IF
END_IF

//Condição de parada do oiclo:
IF NOT xParBStopTankD THEN
	running := FALSE;
	xParBomba1D := FALSE;
	xParBomba2D := FALSE;
	xParBomba3D := FALSE;
	xParAquecD := FALSE;
	xParMistD := FALSE;
	xParRunTankD := FALSE;
	xParFullTankD := FALSE;
	xParIdleD := FALSE;
END_IF

END_PROGRAM

// Device/Application/PROGRAMAS/tanqueA/tanqueA_main
PROGRAM tanqueA_main
VAR
	vmax : INT := REAL_TO_INT((3.1416*((1.5/2)*(1.5/2)))*3.2*1000);
	TIMER : TON;
	conv : REAL :=1;
END_VAR

//Configurações para os blinks:
IF TIMER.Q THEN
	blinkEnable := FALSE;
	blinkTarget := ADR(NULL);
END_IF
TIMER(IN := blinkEnable, PT := REAL_TO_TIME(blinkDuration*1E3));
blinkTarget^ := INT_TO_BOOL(REAL_TO_INT(TIME_TO_REAL(TIMER.ET)/(tonoff*1E3)) MOD 2);

//Associação das entradas analógicas:
rTankALevel := (320.0*iParUltras/27648.0);
iParDisplayNivel := REAL_TO_INT(8192.0*rTankALevel/320.0);
rTankATemp := (100.0*iParTerm/27648.0);
iParDisplayTemp := REAL_TO_INT(8192.0*rTankATemp/100.0);
rTankAVol := (rTankALevel/(VOL_TO_LEVEL(1)*1000));
IF xEnableTankA THEN
	CASE iTankAUnit OF
		1: conv := 1.0; //litros
		2: conv := (1.0/VOL_TO_LEVEL(1)); //centímetros
		3: conv := (vmax/100.0); //porcentagem
	END_CASE
	rTankASP1 := (conv*rSupI1);
	rTankASP2 := (conv*rSupI2);
	rTankASPTemp := rSupT;
	LimTankAConv := (LimTankA/conv);
	capMax := (vmax/conv);
	defaultUnit := iTankAUnit-1;
	IF (NOT xTankARunning) THEN
		processID := 0;
	END_IF
ELSE
	rTankASP1 := (10056.0*iParSPB1/27648.0);
	rTankASP2 := (10056.0*iParSPB2/27648.0);
	rTankASPTemp := (100.0*iParSPTemp/27648.0);
	defaultUnit := 0;
END_IF
IF (rTankALevel<VOL_TO_LEVEL(rTankASP1)) THEN
	offset := rTankALevel;
ELSE
	offset := VOL_TO_LEVEL(rTankASP1);
END_IF

//Condição de parada, segurança, proteção e requisitos mínimos e máximos:
LimTankA := (vmax-rTankASP1);
allowStart := ((rTankASP1>=1000) AND (rTankASP2>=1000) AND (rTankASP1<=vmax) AND (rTankASP2<=LimTankA) AND (rTankASPTemp>=10) AND ((processTarget>0) OR xEndLess OR (TankAMode=1)));
IF rTankALevel >= 320 THEN
	xParBomba1A := FALSE;
	xParBomba2A := FALSE;
END_IF
IF rTankALevel <= 0 THEN
	xParBomba3A := FALSE;
END_IF
//Botoeira de STOP:
IF ((NOT xParBStopTankA) AND (TankAMode <> 3)) THEN
	xTankARunning := FALSE;
	xParBomba1A := FALSE;
	xParBomba2A := FALSE;
	xParBomba3A := FALSE;
	xParAquecA := FALSE;
	xParMistA := FALSE;
	xParRunTankA := FALSE;
	xParFullTankA := FALSE;
	xParIdleA := FALSE;
	blinkEnable := FALSE;
END_IF

//Alerta de condições não satisfeitas:
IF xParBStartTankA THEN
	IF ((NOT allowStart) AND ((TankAMode = 1) OR (TankAMode = 2))) THEN
		//Configura o blink:
		blinkEnable :=TRUE;
		blinkDuration := 3;
		tonoff := 0.5;
		blinkTarget := ADR(xParFullTankA);
		xTankARunning := FALSE;
	ELSE
		IF ((TankAMode <> 0) AND (TankAMode <> 3)) THEN
			xTankARunning := TRUE;
		END_IF		
	END_IF
END_IF

//Verifica chaves da planta e prioriza o supervisório:
IF ((NOT xEnableTankA) AND (NOT halfCicle)) THEN
	IF xParChCTankA THEN
		TankAMode := 3;
	ELSE
			IF xParChATankA THEN
				TankAMode := 1;
			ELSE
				IF xParChBTankA THEN
					TankAMode := 2;
				ELSE
					TankAMode := 0;
					xTankARunning := FALSE;
				END_IF
			END_IF
	END_IF
END_IF

//Seleção do modo de operação:
IF (xTankARunning OR (TankAMode=3)) THEN
	CASE TankAMode OF
		1:	//Batelada:
			tanqueA_process(loop:=FALSE);
			IF(NOT halfCicle) THEN
				xTankARunning := FALSE;
			END_IF
		2:	//Automático:
			tanqueA_process(loop:=TRUE);
		3:	//Modo de manutenção:
			tanqueA_manut();
	END_CASE
END_IF

END_PROGRAM

// Device/Application/PROGRAMAS/tanqueA/VOL_TO_LEVEL
FUNCTION VOL_TO_LEVEL : REAL
VAR_INPUT
	vol : REAL;
END_VAR

VAR
END_VAR

VOL_TO_LEVEL := ((4.0*vol)/(10.0*3.14159*1.5*1.5));

END_FUNCTION

// Device/Application/PROGRAMAS/tanqueA/tanqueA_process
PROGRAM tanqueA_process
VAR
	mixtimer : TON;
	state : INT := 0;
END_VAR

VAR_INPUT
	loop : BOOL;
END_VAR

//Declaração do timer de desligamento da mistura:
mixtimer(IN:=((state=6) AND xTankARunning), PT:=T#5S);


//Condição de início do ciclo:
IF (xParBStartTankA AND allowStart) THEN
	processID := 0;
	IF state = 0 THEN
		IF loop THEN
			state := 1;
		ELSE
			state := 3;
		END_IF		
	END_IF
END_IF

CASE state OF
	1:	//Alerta de início de processo:
		IF (loop AND ((processID < processTarget) OR xEndLess)) THEN
			//Configura o blink:
			blinkEnable := TRUE;
			blinkDuration := 5;
			tonoff := 0.5;
			blinkTArget := ADR(xParIdleA);
		END_IF
		state := 2;
	2:	//Aguarda tempo para início do processo:
		IF NOT blinkEnable THEN
			state := 3;
		END_IF		
	3:	//Indicação de ciclo em andamento:
		halfCicle := TRUE;
		heat := FALSE;
		//Adiciona ingrediente 1
		xParBomba1A := TRUE;
		IF (rTankALevel >= VOL_TO_LEVEL(rTankASP1)) THEN
			xParBomba1A := FALSE;
			state := 4;
		END_IF
	4:	//Adiciona ingrediente 2
		xParBomba2A := TRUE;
		IF ((rTankALevel-VOL_TO_LEVEL(rTankASP1)) >= VOL_TO_LEVEL(rTankASP2)) THEN
			xParBomba2A := FALSE;
			state := 5;
		END_IF
	5: 	//Liga o misturador e o aquecedor e aguarda aquecimento:
		xParMistA := TRUE;
		xParAquecA := TRUE;
		IF (rTankATemp >= rTankASPTemp) THEN
			xParAquecA := FALSE;
			heat := TRUE;
			state := 6;
		END_IF
	6:	//Aguarda o timer e desliga o misturador:
		xParMistA := TRUE;
		IF mixtimer.Q THEN
			xParMistA := FALSE;
			state := 7;
		END_IF
	7:	//Esvazia o tanque:
		xParBomba3A := TRUE;
		IF (rTankALevel = 0) THEN
			xParBomba3A := FALSE;
			//Indicação de ciclo em andamento:
			halfCicle := FALSE;		
			IF loop THEN
				state := 1;
			ELSE
				state := 0;
			END_IF
			//Adiciona resultado à produção total:
			batCont := (batCont+1);
			prod := (prod+rTankASP1+rTankASP2);
			processID := (processID+1);
			IF ((processID = processTarget) AND (NOT xEndLess)) THEN
				xTankARunning := FALSE;
			END_IF
			//Condição de parada após o processo atual:
			IF (xstopAfterCurrent AND (NOT halfCicle)) THEN
				xTankARunning := FALSE;
				xstopAfterCurrent := FALSE;
			END_IF		
		END_IF
END_CASE 

//Indicações pelos sinaleiros da planta:
xParRunTankA := halfCicle;
xParFullTankA := (state>4);
IF NOT blinkEnable THEN
	xParIdleA := (state=7);
END_IF

END_PROGRAM

// Device/Application/PROGRAMAS/tanqueA/tanqueA_manut
PROGRAM tanqueA_manut
VAR
END_VAR

//Aciona bombas de entrada:
IF rTankALevel < 320 THEN
	xParBomba1A := xParBStartTankA;
	xParBomba2A := xParBStartTankA;
	xParRunTankA := xParBStartTankA;
ELSE
	xParBomba1A := FALSE;
	xParBomba2A := FALSE;
	xParRunTankA := FALSE;
END_IF

//Aciona bomba de saída:
IF rTankALevel > 0 THEN
	xParBomba3A := NOT xParBStopTankA;
	xParIdleA := NOT xParBStopTankA;
ELSE
	xParBomba3A := FALSE;
	xParIdleA := FALSE;
END_IF

//Sinalizando condições de contorno:
xParFullTankA := (((rTankALevel >= 320) AND xParBStartTankA) OR ((rTankALevel <= 0) AND (NOT xParBStopTankA)));

END_PROGRAM

// Device/Application/Visualizations/tanque_DIG
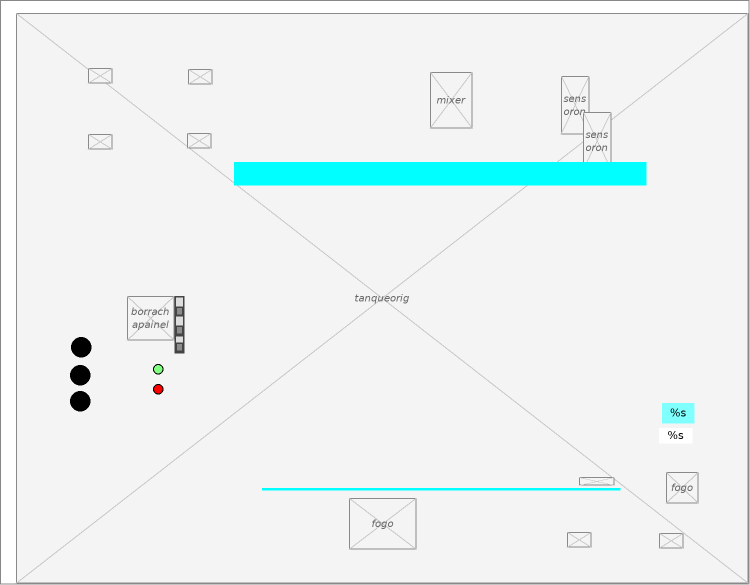
VISUALIZATION tanque_DIG  // 750x585
    Image (16,13 732x570), image: tanqueorig
    Rectangle (262,488 358x2), invisible if: SIM_TANQUE_DIG.nivelCM=0
        p2773130477: SIM_TANQUE_DIG.nivelCM*-1
    Image (561,76 28x58), invisible if: NOT .xParAltoD, image: sensoron
    Image (583,112 28x58), invisible if: NOT .xParBaixoD, image: sensoron
    Image (88,134 24x15), invisible if: NOT SIM_TANQUE_DIG.PF2, image: sensorfluxo
    Image (88,68 24x15), invisible if: NOT SIM_TANQUE_DIG.PF1, image: sensorfluxo
    Image (567,532 24x15), invisible if: NOT SIM_TANQUE_DIG.PF3, image: sensorfluxo
    Ellipse (153,364 10x10)
        tap .xParBStartTankD
    Ellipse (153,384 10x10)
        tap .xParBStopTankD p1329445385=TRUE
    Ellipse (71,337 20x20), colour toggle: .xParRunTankD
    Ellipse (70,365 20x20), colour toggle: .xParIdleD
    Ellipse (70,391 20x20), colour toggle: .xParFullTankD
    Image (349,498 67x51), invisible if: NOT SIM_TANQUE_DIG.PFIRE, image: fogo
    Image (430,72 42x56), invisible if: NOT SIM_TANQUE_DIG.MIX1, image: mixer
    Rectangle (662,403 32x20), "%s", text variable: SIM_TANQUE_DIG.tempadj
        OnMouseDown: write the text variable via VisuDialogs.Numpad, min 0, max 100
    Rectangle (659,428 33x15), "%s", text variable: SIM_TANQUE_DIG.cchama.CV, colour toggle: SIM_TANQUE_DIG.cchama.CV >= SIM_TANQUE_DIG.tempadj
    Image (579,477 35x8), invisible if: SIM_TANQUE_DIG.cchama.CV < SIM_TANQUE_DIG.tempadj, image: termo
    Image (666,472 32x31), invisible if: NOT SIM_TANQUE_DIG.bombafogo, image: fogo
    Rectangle (234,162 412x23), invisible if: SIM_TANQUE_DIG.nivelCM<=320
        p1126004900: SIM_TANQUE_DIG.CTRANSB.CV*5
    Image (127,296 47x44), image: borrachapainel
    Image (188,69 24x15), invisible if: NOT SIM_TANQUE_DIG.PF1, image: sensorfluxo
    Image (187,133 24x15), invisible if: NOT SIM_TANQUE_DIG.PF2, image: sensorfluxo
    Image (659,533 24x15), invisible if: NOT SIM_TANQUE_DIG.PF3, image: sensorfluxo
    DipSwitch (169,328 21x29), variable: xParChCTankD, behaviour: TOGGLE, style: Switch-DipSwitch-Gray
    DipSwitch (169,292 21x29), variable: xParChATankD, behaviour: TOGGLE, style: Switch-DipSwitch-Gray
    DipSwitch (169,311 21x29), variable: xParChBTankD, behaviour: TOGGLE, style: Switch-DipSwitch-Gray
END_VISUALIZATION

// Device/Application/Visualizations/SILO
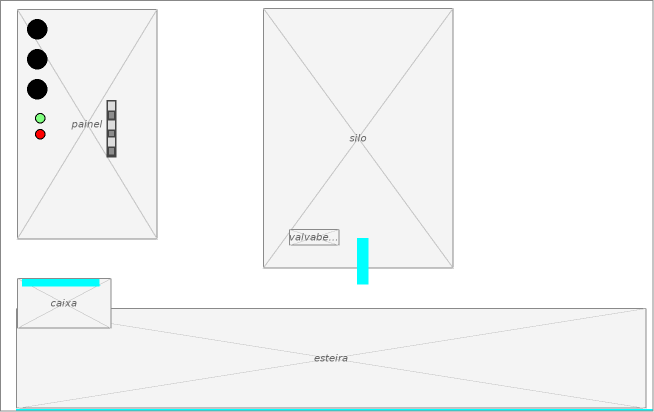
VISUALIZATION SILO  // 654x412
    Group (16,8 636x402)
        Image (1,1 140x230), image: painel
        Image (247,0 190x260), image: silo
        Image (0,300 630x100), image: esteira
        Image (1,270 94x50), image: caixa
            p3560616238: SIM_SILO.caixa_mov
        Rectangle (409,349 7x16), colour toggle: .xParProx, invisible if: NOT .xParProx
        Rectangle (0,401 636x1), invisible if: SIM_SILO.alaga=0
            p2773130477: -SIM_SILO.alaga
        Image (273,221 50x16), invisible if: NOT .xParValve, image: valvaberta
        Ellipse (19,105 10x10)
            tap .xParBStartSilo
        Ellipse (19,121 10x10)
            tap .xParBStopSilo p1329445385=TRUE
        Ellipse (11,11 20x20), colour toggle: .xParRunSilo
        Ellipse (11,41 20x20), colour toggle: .xParFillSilo
        Ellipse (11,71 20x20), colour toggle: .xParFullSilo
        Rectangle (371,212 7x26), colour toggle: .xParLevel, invisible if: NOT .xParLevel
        Rectangle (341,230 11x46), invisible if: NOT .xParValve
        DipSwitch (85,88 21x29), variable: xParChASilo, behaviour: TOGGLE, style: Switch-DipSwitch-Gray
        DipSwitch (85,107 21x29), variable: xParChBSilo, behaviour: TOGGLE, style: Switch-DipSwitch-Gray
        DipSwitch (85,124 21x29), variable: xParChCSilo, behaviour: TOGGLE, style: Switch-DipSwitch-Gray
        Rectangle (7,277 77x0), invisible if: SIM_SILO.clevel.CV<24
            p3560616238: SIM_SILO.caixa_mov
            p2773130477: -SIM_SILO.clevel.CV+24
        Rectangle (6,271 77x7), invisible if: NOT SIM_SILO.CHEIA
            p3560616238: SIM_SILO.caixa_mov
END_VISUALIZATION

// Device/Application/Visualizations/semaforo
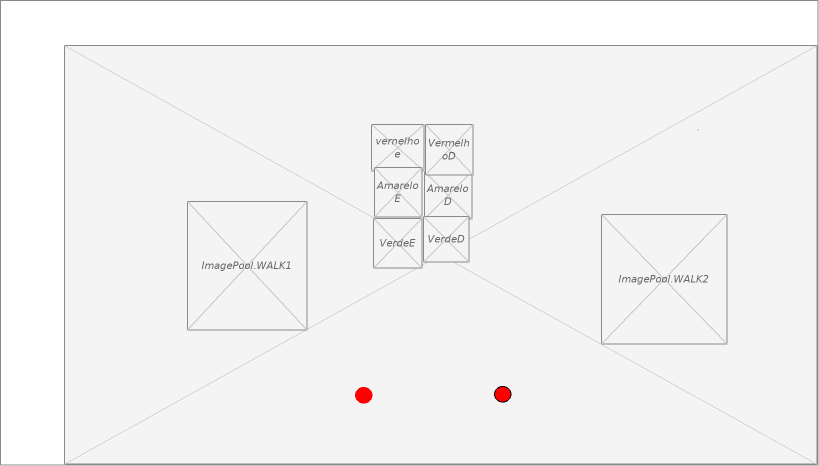
VISUALIZATION semaforo  // 819x466
    Image (64,45 753x419), image: semaforo
    Image (371,124 53x47), invisible if: NOT xParafVermE, image: vernelhoe
    Image (424,171 48x48), invisible if: NOT xParafAmarD, image: AmareloD
    Image (373,218 49x50), invisible if: NOT xParafVerdE, image: VerdeE
    Image (425,124 48x51), invisible if: NOT .xParafVermD, image: VermelhoD
    Image (374,167 48x50), invisible if: NOT xParafAmarE, image: AmareloE
    Image (423,216 46x46), invisible if: NOT .xParafVerdD, image: VerdeD
    Ellipse (494,386 17x16)
        tap xParafBPedD
    Ellipse (355,387 17x16)
        tap xParafBPedE
    Image (187,201 120x129), image: ImagePool.WALK1
    Image (601,214 126x130), image: ImagePool.WALK2
    Image (698,129 0x1), image: ImagePool.WALK2
END_VISUALIZATION

// Device/Application/Visualizations/garagem
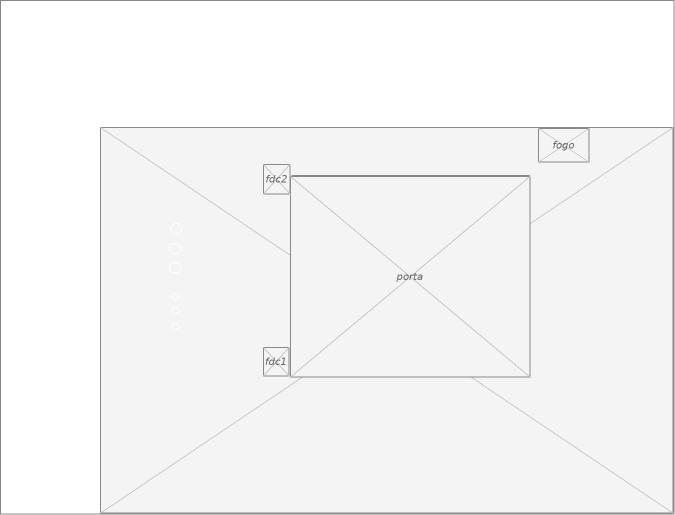
VISUALIZATION garagem  // 675x515
    Group (100,127 573x386)
        Image (0,0 573x386), image: garagem
        Image (191,48 239x199), image: onibus
        Image (190,49 240x201), image: porta
            p1126004900: -.SIM_GARAGEM.porta
        Image (163,220 26x29), invisible if: .xParLs2, image: fdc1
        Image (163,37 27x30), invisible if: .xParLs1, image: fdc2
        Image (438,1 51x34), invisible if: NOT SIM_GARAGEM.fogo, image: fogo
        Ellipse (70,96 12x11), colour toggle: .xParAjar
        Ellipse (69,116 12x11), colour toggle: .xParOpen
        Ellipse (69,135 12x11), colour toggle: .xParShut
        Ellipse (72,166 7x7)
            tap .xParBOpen
        Ellipse (72,180 7x7)
            tap .xParBClose
        Ellipse (72,196 7x7)
            tap .xParBStopGar p1329445385=TRUE
        Rectangle (448,32 6x17), colour toggle: (SIM_GARAGEM.Pisca ) <> 0, invisible if: NOT .xParMotorUp
        Rectangle (457,31 6x17), colour toggle: (SIM_GARAGEM.Pisca ) <> 0, invisible if: NOT .xParMotorDown
END_VISUALIZATION

// Device/Application/Visualizations/tanque_ANALOG
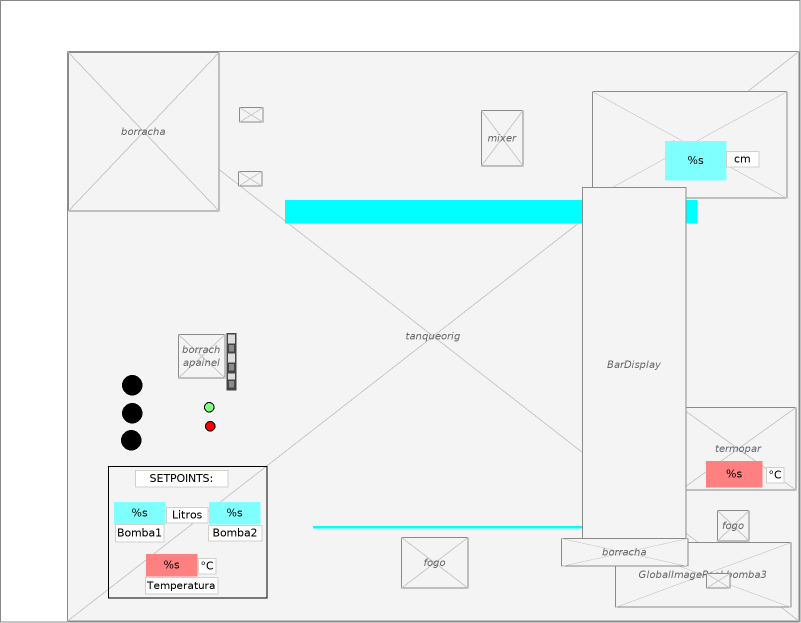
VISUALIZATION tanque_ANALOG  // 801x623
    Image (67,51 732x570), image: tanqueorig
    Rectangle (108,466 159x132)
    Rectangle (313,526 358x2), invisible if: SIM_TANQUE_ANALOG.nivelCM=0
        p2773130477: SIM_TANQUE_ANALOG.nivelCM*-1
    Ellipse (204,402 10x10)
        tap .xParBStartTankA
    Ellipse (205,421 10x10)
        tap .xParBStopTankA p1329445385=TRUE
    Ellipse (122,375 20x20), colour toggle: .xParRunTankA
    Ellipse (122,403 20x20), colour toggle: .xParIdleA
    Ellipse (121,430 20x20), colour toggle: .xParFullTankA
    Image (401,537 67x51), invisible if: not xParAquecA, image: fogo
    Image (481,110 42x56), invisible if: NOT SIM_TANQUE_ANALOG.MIX1, image: mixer
    Image (717,510 32x31), invisible if: NOT SIM_TANQUE_ANALOG.bombafogo, image: fogo
    Rectangle (285,200 412x23), invisible if: SIM_TANQUE_ANALOG.nivelCM<=320
        p1126004900: SIM_TANQUE_ANALOG.CTRANSB.CV*5
    Image (178,334 47x44), image: borrachapainel
    Image (239,107 24x15), invisible if: NOT SIM_TANQUE_ANALOG.PF1, image: sensorfluxo
    Image (238,171 24x15), invisible if: NOT SIM_TANQUE_ANALOG.PF2, image: sensorfluxo
    Image (592,91 195x107), tooltip "0 a 10 mV", image: ultrassom
    Image (680,407 116x83), tooltip "4 a 20 mA", image: termopar
    Image (68,52 151x159), image: borracha
    BarDisplay (582,187 104x355), value: SIM_TANQUE_ANALOG.nivelCM, scale format: %.1f, scale 0..320
    Rectangle (114,502 51x22), "%s", text variable: .SIM_TANQUE_ANALOG.setbomba1
        OnMouseDown: write the text variable via InputWithLimits, min 0, max 10056
    Rectangle (209,502 51x22), "%s", text variable: .SIM_TANQUE_ANALOG.setbomba2
        OnMouseDown: write the text variable via InputWithLimits, min 0, max 10056
    Textfield (115,524 49x18), "Bomba1"
    Textfield (208,525 54x16), "Bomba2"
    Rectangle (665,141 61x39), "%s", text variable: iParDisplayNivel*320/8192
    Rectangle (706,461 56x26), "%s", text variable: iParDisplayTemp*100/8192
    Textfield (135,470 93x17), "SETPOINTS:"
    Textfield (145,577 73x17), "Temperatura"
    Rectangle (146,554 51x22), "%s", text variable: .SIM_TANQUE_ANALOG.settemp
        OnMouseDown: write the text variable via InputWithLimits, min 0, max 100
    Textfield (166,507 42x16), "Litros"
    Textfield (198,558 18x16), "°C"
    Textfield (766,467 18x16), "°C"
    Textfield (726,151 33x16), "cm"
    Image (615,542 176x65), image: GlobalImagePool.bomba3
    Image (561,538 127x28), image: borracha
    DipSwitch (221,365 21x29), variable: xParChCTankA, behaviour: TOGGLE, style: Switch-DipSwitch-Gray
    DipSwitch (221,329 21x29), variable: xParChATankA, behaviour: TOGGLE, style: Switch-DipSwitch-Gray
    DipSwitch (221,348 21x29), variable: xParChBTankA, behaviour: TOGGLE, style: Switch-DipSwitch-Gray
    Image (706,573 24x15), invisible if: NOT SIM_TANQUE_ANALOG.PF3, image: sensorfluxo
END_VISUALIZATION
